// TwinCAT 3 PLC project Untitled1
// ProgramVersion: 3.1.4023.0
// libraries:
//   Tc2_Standard, * (Beckhoff Automation GmbH)
//   Tc2_System, * (Beckhoff Automation GmbH)
//   Tc3_Module, * (Beckhoff Automation GmbH)
// project tree:
//   / PlcTask.TcTTO
//   POUs/ FB_ClkSignal.TcPOU, MAIN.TcPOU
// real-time tasks:
//   TASK PlcTask: cycle T#10ms, priority 20, ADS port 350

CONFIGURATION Untitled1
    RESOURCE PLC ON TwinCAT3
        TASK PlcTask(INTERVAL := T#10ms, PRIORITY := 20);
        PROGRAM MAIN WITH PlcTask : MAIN;
    END_RESOURCE
END_CONFIGURATION

// ---- POUs/MAIN.TcPOU
PROGRAM MAIN
VAR
	FB_ClkSignal_1	:	FB_ClkSignal;
END_VAR

FB_ClkSignal_1(IN_bStart:= , IN_fFrequency:=0.001 , OUT_Signal=> );

END_PROGRAM

// ---- POUs/FB_ClkSignal.TcPOU
FUNCTION_BLOCK FB_ClkSignal
VAR_INPUT
	IN_bStart: BOOL;
	IN_fFrequency: REAL;
END_VAR
VAR_OUTPUT
	OUT_Signal: BOOL;
END_VAR
VAR
	nState: INT;
	TON1: TON;
	TON2: TON;
	tTime: TIME;
END_VAR

tTime := REAL_TO_TIME(1/IN_fFrequency);

CASE nState OF
	
0:

	IF IN_bStart THEN
		
		nState := 10;
		
	END_IF

10:

	TON1(IN:= TRUE , PT:= tTime , Q=> , ET=> );	
	OUT_Signal	:=	FALSE;
	
	IF TON1.Q THEN

		nState	:= 20;	
		TON1(IN:=FALSE);

	END_IF
	
20:

	TON2(IN:= TRUE , PT:=tTime , Q=> , ET=> );
	OUT_Signal	:=	TRUE;
	
	IF TON2.Q THEN

		nState	:= 0;	
		TON2(IN:=FALSE);
		
	END_IF

END_CASE

END_FUNCTION_BLOCK
